// Mitsubishi GX Works2 project: 12   PLC: Q03UDV

PROGRAM MAIN
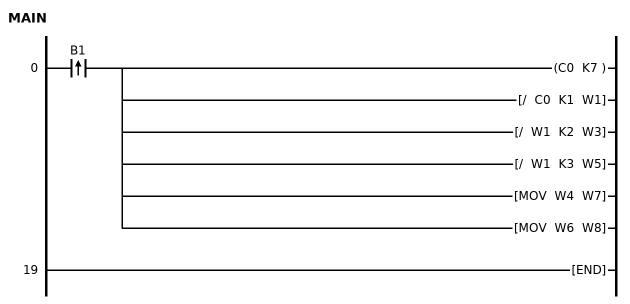
0     LDP     B1
      OUT     C0 K7
      /       C0 K1 W1
      /       W1 K2 W3
      /       W1 K3 W5
      MOV     W4 W7
      MOV     W6 W8
19    END
END_PROGRAM
